// LS Electric XG5000 project: 120대대(250508)
// PLC NewPLC
// module base 0 slot 0: 16점 예약 할당:XG-IN16
// module base 0 slot 1: Cnet:XGL-CH2A/B (Cnet 통신 모듈(RS-232C, RS-422/485))
// module base 0 slot 2: 아날로그입력 모듈:XGF-AC8A (A/D 전류 입력형 8채널)
// module base 0 slot 3: 입력 모듈:XGI-D24A/B (DC 24V 입력, 32점 (전류소스 싱크공용/ 전류소스 입력))
// module base 0 slot 4: 출력 모듈:XGQ-TR4A/B (트랜지스터 출력, 32점 (0.1A용, 싱크출력/소스출력))
// module base 0 slot 5: 고속카운터 모듈:XGF-HO2A (고속카운터 펄스(OC) 입력형, 2채널)

PROGRAM Sequence_Program (task: 스캔 프로그램)

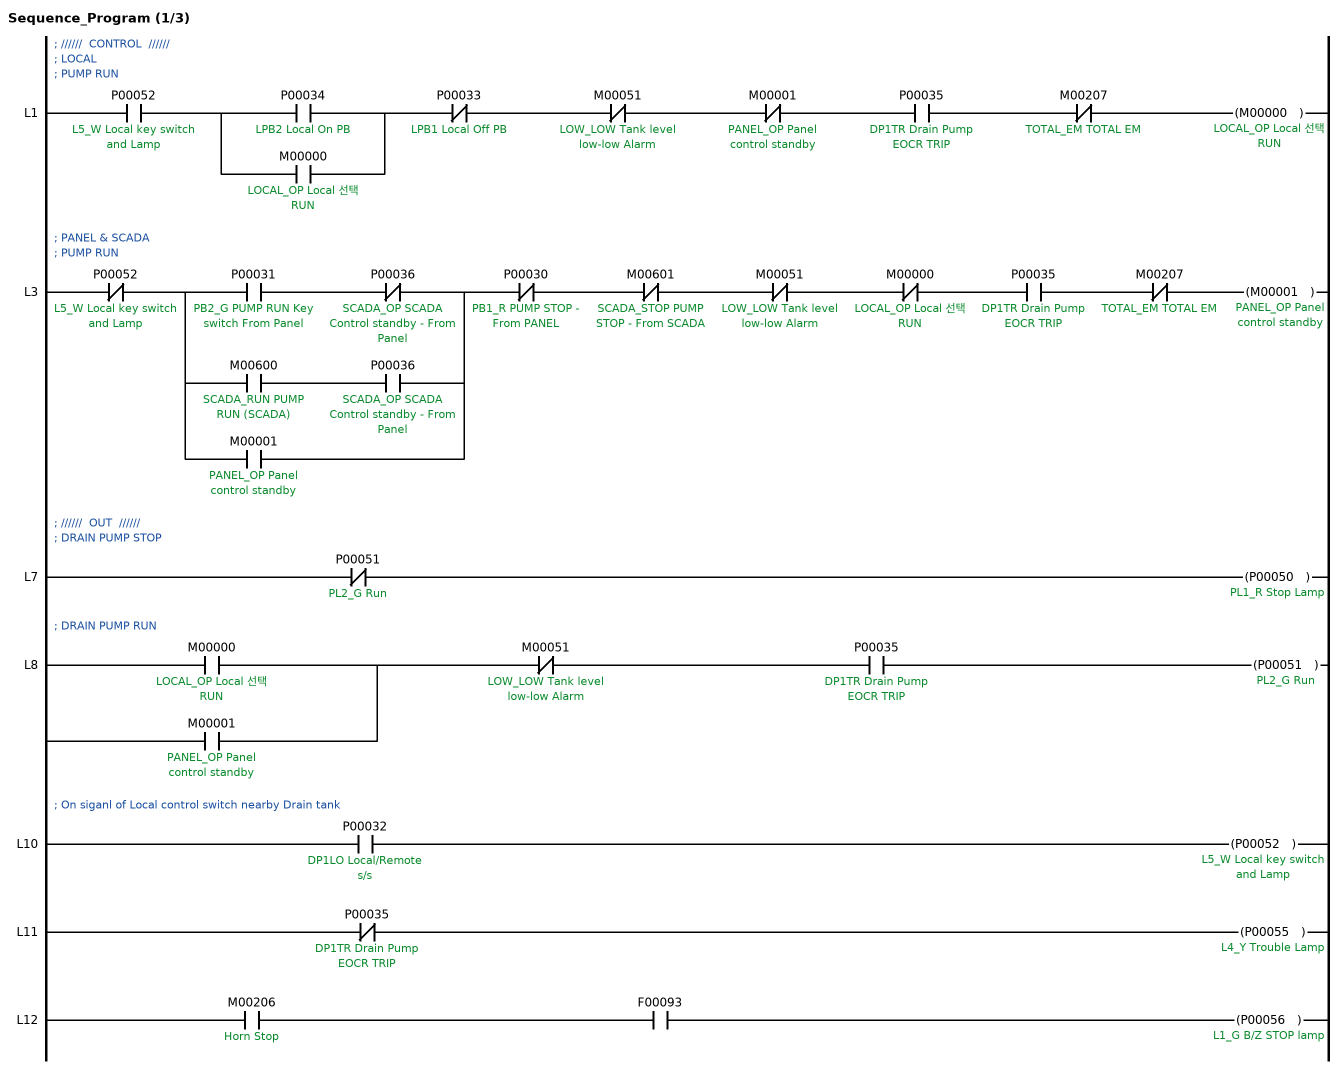
//      //////  CONTROL  //////
; L1
LOAD      P00052	// L5_W Local key switch and Lamp
LOAD      P00034	// LPB2 Local On PB
OR        M00000	// LOCAL_OP Local 선택 RUN
AND LOAD
AND NOT   P00033	// LPB1 Local Off PB
AND NOT   M00051	// LOW_LOW Tank level low-low Alarm
AND NOT   M00001	// PANEL_OP Panel control standby
AND       P00035	// DP1TR Drain Pump EOCR TRIP
AND NOT   M00207	// TOTAL_EM TOTAL EM
OUT       M00000	// LOCAL_OP Local 선택 RUN
// output comment: LOCAL PUMP RUN
; L3
LOAD NOT  P00052	// L5_W Local key switch and Lamp
LOAD      P00031	// PB2_G PUMP RUN Key switch From Panel
AND NOT   P00036	// SCADA_OP SCADA Control standby - From Panel
LOAD      M00600	// SCADA_RUN PUMP RUN (SCADA)
AND       P00036	// SCADA_OP SCADA Control standby - From Panel
OR LOAD
OR        M00001	// PANEL_OP Panel control standby
AND LOAD
AND NOT   P00030	// PB1_R PUMP STOP - From PANEL
AND NOT   M00601	// SCADA_STOP PUMP STOP - From SCADA
AND NOT   M00051	// LOW_LOW Tank level low-low Alarm
AND NOT   M00000	// LOCAL_OP Local 선택 RUN
AND       P00035	// DP1TR Drain Pump EOCR TRIP
AND NOT   M00207	// TOTAL_EM TOTAL EM
OUT       M00001	// PANEL_OP Panel control standby
// output comment: PANEL & SCADA PUMP RUN
//      //////  OUT  //////
; L7
LOAD NOT  P00051	// PL2_G Run
OUT       P00050	// PL1_R Stop Lamp
// output comment: DRAIN PUMP STOP
; L8
LOAD      M00000	// LOCAL_OP Local 선택 RUN
OR        M00001	// PANEL_OP Panel control standby
AND NOT   M00051	// LOW_LOW Tank level low-low Alarm
AND       P00035	// DP1TR Drain Pump EOCR TRIP
OUT       P00051	// PL2_G Run
// output comment: DRAIN PUMP RUN
; L10
LOAD      P00032	// DP1LO Local/Remote s/s
OUT       P00052	// L5_W Local key switch and Lamp
// output comment: On siganl of Local control switch nearby Drain tank
; L11
LOAD NOT  P00035	// DP1TR Drain Pump EOCR TRIP
OUT       P00055	// L4_Y Trouble Lamp
// output comment: 
; L12
LOAD      M00206	// Horn Stop
AND       F00093
OUT       P00056	// L1_G B/Z STOP lamp
// output comment: 

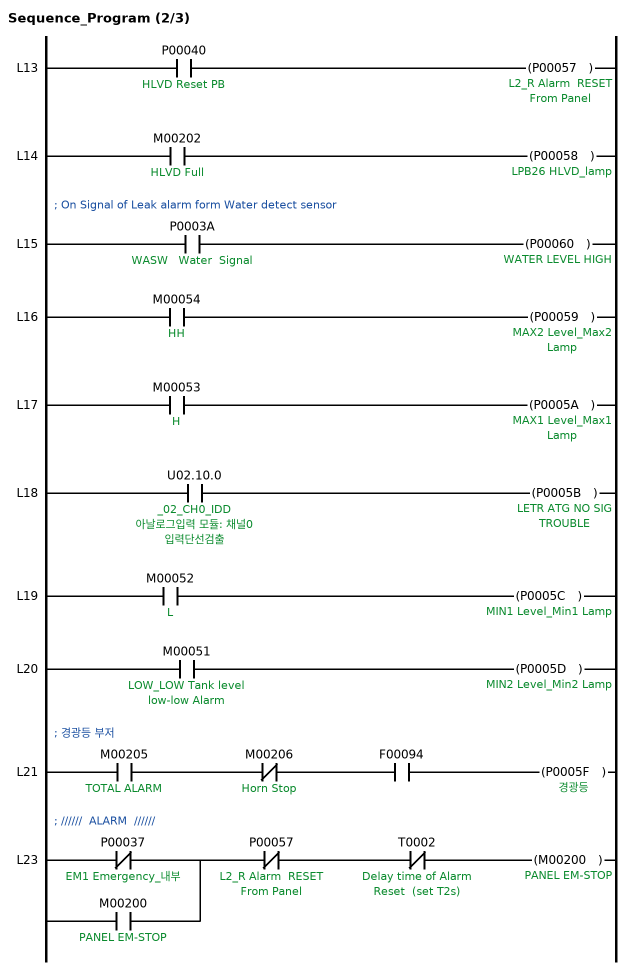
; L13
LOAD      P00040	// HLVD Reset PB
OUT       P00057	// L2_R Alarm  RESET From Panel
// output comment: 
; L14
LOAD      M00202	// HLVD Full
OUT       P00058	// LPB26 HLVD_lamp
; L15
LOAD      P0003A	// WASW   Water  Signal
OUT       P00060	// WATER LEVEL HIGH
// output comment: On Signal of Leak alarm form Water detect sensor
; L16
LOAD      M00054	// HH
OUT       P00059	// MAX2 Level_Max2 Lamp
; L17
LOAD      M00053	// H
OUT       P0005A	// MAX1 Level_Max1 Lamp
; L18
LOAD      U02.10.0	// _02_CH0_IDD 아날로그입력 모듈: 채널0 입력단선검출
OUT       P0005B	// LETR ATG NO SIG TROUBLE
; L19
LOAD      M00052	// L
OUT       P0005C	// MIN1 Level_Min1 Lamp
; L20
LOAD      M00051	// LOW_LOW Tank level low-low Alarm
OUT       P0005D	// MIN2 Level_Min2 Lamp
; L21
LOAD      M00205	// TOTAL ALARM
AND NOT   M00206	// Horn Stop
AND       F00094
OUT       P0005F	// 경광등
// output comment: 경광등 부저
//      //////  ALARM  //////
; L23
LOAD NOT  P00037	// EM1 Emergency_내부
OR        M00200	// PANEL EM-STOP
AND NOT   P00057	// L2_R Alarm  RESET From Panel
AND NOT   T0002	// Delay time of Alarm Reset  (set T2s)
OUT       M00200	// PANEL EM-STOP

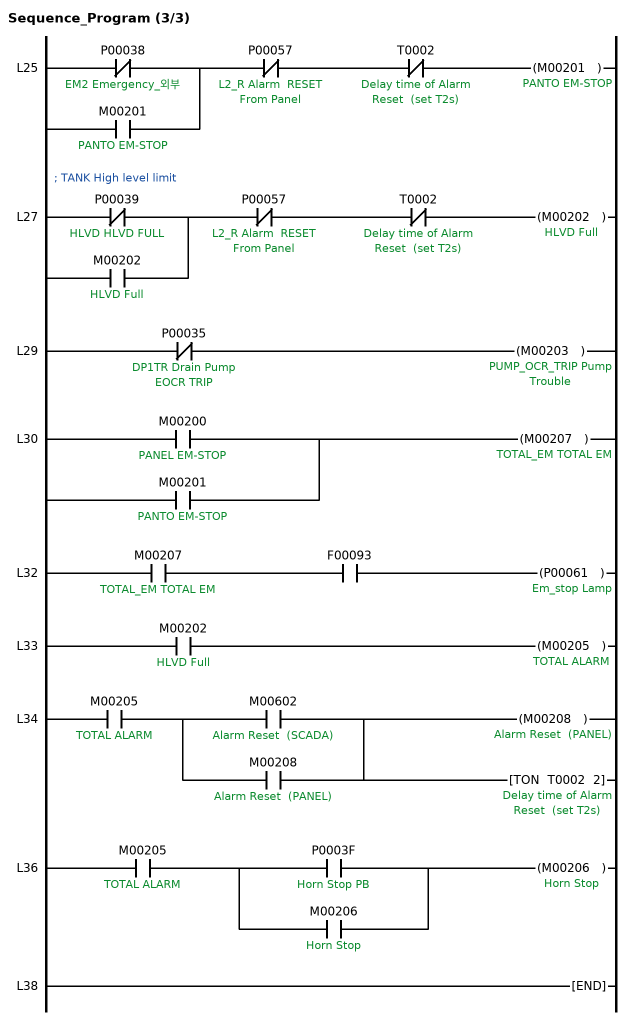
; L25
LOAD NOT  P00038	// EM2 Emergency_외부
OR        M00201	// PANTO EM-STOP
AND NOT   P00057	// L2_R Alarm  RESET From Panel
AND NOT   T0002	// Delay time of Alarm Reset  (set T2s)
OUT       M00201	// PANTO EM-STOP
; L27
LOAD NOT  P00039	// HLVD HLVD FULL
OR        M00202	// HLVD Full
AND NOT   P00057	// L2_R Alarm  RESET From Panel
AND NOT   T0002	// Delay time of Alarm Reset  (set T2s)
OUT       M00202	// HLVD Full
// output comment: TANK High level limit
; L29
LOAD NOT  P00035	// DP1TR Drain Pump EOCR TRIP
OUT       M00203	// PUMP_OCR_TRIP Pump Trouble
; L30
LOAD      M00200	// PANEL EM-STOP
OR        M00201	// PANTO EM-STOP
OUT       M00207	// TOTAL_EM TOTAL EM
; L32
LOAD      M00207	// TOTAL_EM TOTAL EM
AND       F00093
OUT       P00061	// Em_stop Lamp
; L33
LOAD      M00202	// HLVD Full
OUT       M00205	// TOTAL ALARM
; L34
LOAD      M00205	// TOTAL ALARM
LOAD      M00602	//   Alarm Reset  (SCADA)
OR        M00208	//  Alarm Reset  (PANEL)
AND LOAD
OUT       M00208	//  Alarm Reset  (PANEL)
TON       T0002 2	// Delay time of Alarm Reset  (set T2s)
; L36
LOAD      M00205	// TOTAL ALARM
LOAD      P0003F	// Horn Stop PB
OR        M00206	// Horn Stop
AND LOAD
OUT       M00206	// Horn Stop
; L38
END

PROGRAM Analog (task: 스캔 프로그램)

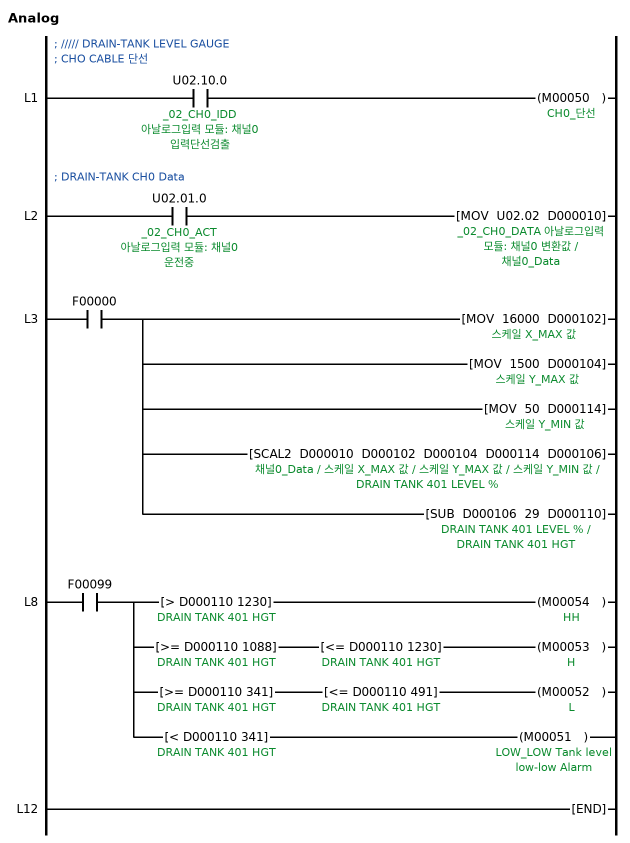
// ///// DRAIN-TANK LEVEL GAUGE
; L1
LOAD      U02.10.0	// _02_CH0_IDD 아날로그입력 모듈: 채널0 입력단선검출
OUT       M00050	// CH0_단선
// output comment: CHO CABLE 단선
; L2
LOAD      U02.01.0	// _02_CH0_ACT 아날로그입력 모듈: 채널0 운전중
MOV       U02.02 D000010	// _02_CH0_DATA 아날로그입력 모듈: 채널0 변환값 / 채널0_Data
// output comment: DRAIN-TANK CH0 Data
; L3
LOAD      F00000
MOV       16000 D000102	// 스케일 X_MAX 값
MOV       1500 D000104	// 스케일 Y_MAX 값
MOV       50 D000114	// 스케일 Y_MIN 값
SCAL2     D000010 D000102 D000104 D000114 D000106	// 채널0_Data / 스케일 X_MAX 값 / 스케일 Y_MAX 값 / 스케일 Y_MIN 값 / DRAIN TANK 401 LEVEL %
SUB       D000106 29 D000110	// DRAIN TANK 401 LEVEL % / DRAIN TANK 401 HGT
; L8
LOAD      F00099
MPUSH
AND>      D000110 1230	// DRAIN TANK 401 HGT
OUT       M00054	// HH
MLOAD
AND>=     D000110 1088	// DRAIN TANK 401 HGT
AND<=     D000110 1230	// DRAIN TANK 401 HGT
OUT       M00053	// H
MLOAD
AND>=     D000110 341	// DRAIN TANK 401 HGT
AND<=     D000110 491	// DRAIN TANK 401 HGT
OUT       M00052	// L
MPOP
AND<      D000110 341	// DRAIN TANK 401 HGT
OUT       M00051	// LOW_LOW Tank level low-low Alarm
; L12
END

PROGRAM Modbus-RTU_Comm (task: 스캔 프로그램)

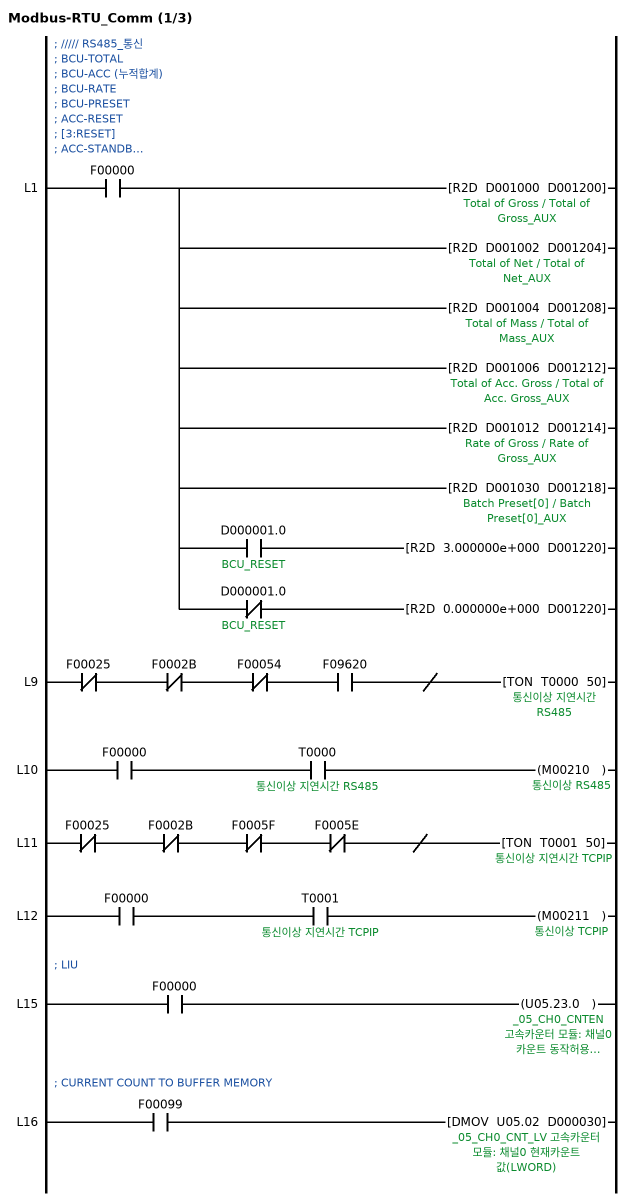
// ///// RS485_통신
; L1
LOAD      F00000
R2D       D001000 D001200	// Total of Gross / Total of Gross_AUX
R2D       D001002 D001204	// Total of Net / Total of Net_AUX
R2D       D001004 D001208	// Total of Mass / Total of Mass_AUX
R2D       D001006 D001212	// Total of Acc. Gross / Total of Acc. Gross_AUX
R2D       D001012 D001214	// Rate of Gross / Rate of Gross_AUX
R2D       D001030 D001218	// Batch Preset[0] / Batch Preset[0]_AUX
MPUSH
AND       D000001.0	// BCU_RESET
R2D       3.000000e+000 D001220
MPOP
AND NOT   D000001.0	// BCU_RESET
R2D       0.000000e+000 D001220
// output comment: BCU-TOTAL
// output comment: BCU-ACC (누적합계)
// output comment: BCU-RATE
// output comment: BCU-PRESET
// output comment: ACC-RESET [3:RESET]
// output comment: ACC-STANDBY [0:STANDBY]
; L9
LOAD NOT  F00025
AND NOT   F0002B
AND NOT   F00054
AND       F09620
NOT
TON       T0000 50	// 통신이상 지연시간 RS485
; L10
LOAD      F00000
AND       T0000	// 통신이상 지연시간 RS485
OUT       M00210	// 통신이상 RS485
; L11
LOAD NOT  F00025
AND NOT   F0002B
AND NOT   F0005F
AND NOT   F0005E
NOT
TON       T0001 50	// 통신이상 지연시간 TCPIP
; L12
LOAD      F00000
AND       T0001	// 통신이상 지연시간 TCPIP
OUT       M00211	// 통신이상 TCPIP
//  LIU
; L15
LOAD      F00000
OUT       U05.23.0	// _05_CH0_CNTEN 고속카운터 모듈: 채널0 카운트 동작허용(Level)지령
; L16
LOAD      F00099
DMOV      U05.02 D000030	// _05_CH0_CNT_LV 고속카운터 모듈: 채널0 현재카운트 값(LWORD)
// output comment: CURRENT COUNT TO BUFFER MEMORY

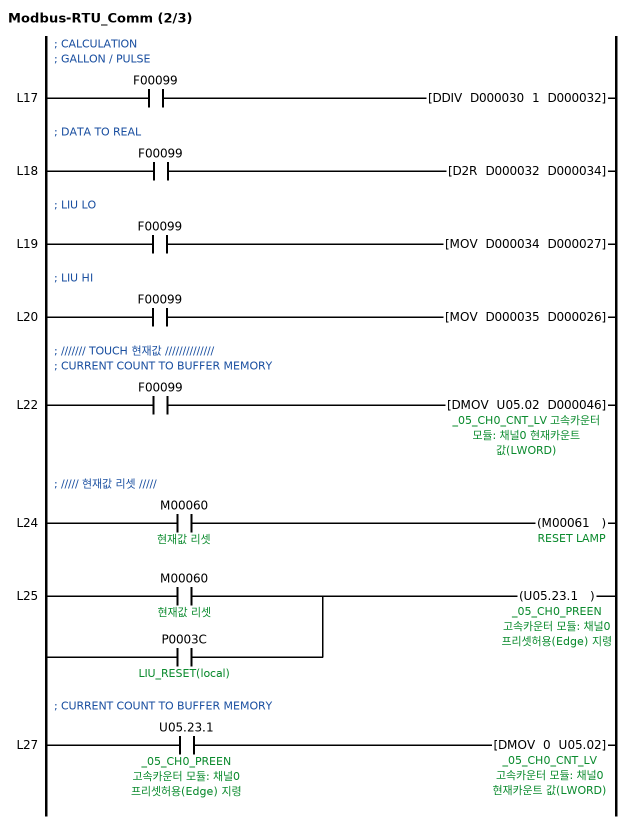
; L17
LOAD      F00099
DDIV      D000030 1 D000032
// output comment: CALCULATION GALLON / PULSE
; L18
LOAD      F00099
D2R       D000032 D000034
// output comment: DATA TO REAL
; L19
LOAD      F00099
MOV       D000034 D000027
// output comment: LIU LO
; L20
LOAD      F00099
MOV       D000035 D000026
// output comment: LIU HI
// /////// TOUCH 현재값 //////////////
; L22
LOAD      F00099
DMOV      U05.02 D000046	// _05_CH0_CNT_LV 고속카운터 모듈: 채널0 현재카운트 값(LWORD)
// output comment: CURRENT COUNT TO BUFFER MEMORY
// ///// 현재값 리셋 /////
; L24
LOAD      M00060	// 현재값 리셋
OUT       M00061	// RESET LAMP
; L25
LOAD      M00060	// 현재값 리셋
OR        P0003C	// LIU_RESET(local)
OUT       U05.23.1	// _05_CH0_PREEN 고속카운터 모듈: 채널0 프리셋허용(Edge) 지령
; L27
LOAD      U05.23.1	// _05_CH0_PREEN 고속카운터 모듈: 채널0 프리셋허용(Edge) 지령
DMOV      0 U05.02	// _05_CH0_CNT_LV 고속카운터 모듈: 채널0 현재카운트 값(LWORD)
// output comment: CURRENT COUNT TO BUFFER MEMORY

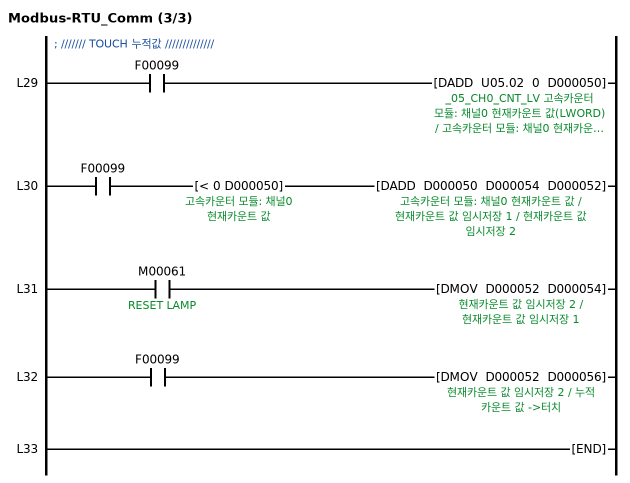
// /////// TOUCH 누적값 //////////////
; L29
LOAD      F00099
DADD      U05.02 0 D000050	// _05_CH0_CNT_LV 고속카운터 모듈: 채널0 현재카운트 값(LWORD) / 고속카운터 모듈: 채널0 현재카운트 값
; L30
LOAD      F00099
AND<      0 D000050	// 고속카운터 모듈: 채널0 현재카운트 값
DADD      D000050 D000054 D000052	// 고속카운터 모듈: 채널0 현재카운트 값 / 현재카운트 값 임시저장 1 / 현재카운트 값 임시저장 2
; L31
LOAD      M00061	// RESET LAMP
DMOV      D000052 D000054	// 현재카운트 값 임시저장 2 / 현재카운트 값 임시저장 1
; L32
LOAD      F00099
DMOV      D000052 D000056	// 현재카운트 값 임시저장 2 / 누적 카운트 값 ->터치
; L33
END

VARIABLES AND COMMENTS (devices not used above)
M0032	WORD	CURR_GALLON
M0034	WORD	CURR_GAL_REAL
M0030	WORD	CURR_PULSE
M00040	BIT	CURR_RST_SIG
M0080	WORD	ERR_CODE
P00041	BIT	LIU_RST_PB
P00053	BIT	LPL1 // DP1-Local Off lamp
P00054	BIT	LPL2 // DP1-Local Run lamp
M0070	WORD	PARITY_ER
M00042	BIT	TOTAL_RST_SIG
D00040.0	BIT	TOTAL_RST_TOUCH
M0062	WORD	국번
M0063	WORD	데이터비트
M0071	WORD	모듈리셋
M0068	WORD	문자간_대기시간
M0064	WORD	스톱비트
M0066	WORD	응답대기시간
M0069	WORD	종단저항
M0067	WORD	지연시간
M0061	WORD	통신속도
M0060	WORD	통신형태
M0065	WORD	페리티
P0003D	BIT	GOCR
D00108	WORD	DRAIN TANK 401 VOL
M00603	BIT	Horn Stop (SCADA)
M00209	BIT	TOTAL ALARM
P0003E	BIT	TLV
D00112	WORD	스케일 X_MIN 값